(* PLC project Unnamed, Unknown Unnamed 1 *)
(* stored: creationDateTime 2022-09-05T09:02:48, modificationDateTime 2022-09-09T09:39:37 *)

FUNCTION_BLOCK my_functionBlock
  VAR
    MYNODE : HMI_NODE;  (* Using HMI_NODE creates node un HMI tree *)
    SOME_INT : HMI_INT;
  END_VAR
  VAR_INPUT
    SOME_STRING : HMI_STRING;
  END_VAR
  VAR
    SOME_BOOL : HMI_BOOL;
    SOME_REAL : HMI_REAL;
  END_VAR
  VAR_INPUT
    SOME_INPUT : BOOL;
  END_VAR
  VAR_OUTPUT
    SOME_OUTPUT : BOOL;
  END_VAR

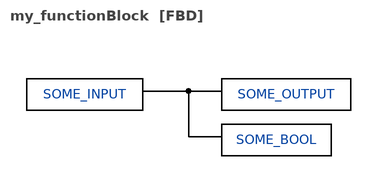
(* FBD diagram, written out as Structured Text *)
SOME_OUTPUT := SOME_INPUT;
SOME_BOOL := SOME_INPUT;
END_FUNCTION_BLOCK

PROGRAM program0
  VAR
    LOGGER0 : LOGGER;
    ENTERING_PAGE : HMI_BOOL;
    LEVEL : LOGLEVEL := DEBUG;
  END_VAR
  VAR_EXTERNAL
    CURRENT_PAGE_0 : HMI_STRING;
  END_VAR
  VAR
    R_TRIG0 : R_TRIG;
    ENABLE_JUMP : HMI_BOOL;
    FB_ZERO : my_functionBlock;
    FB_ONE : my_functionBlock;
    FB_TWO : my_functionBlock;
    FB_THREE : my_functionBlock;
    FB_FOUR : my_functionBlock;
    FB_FIVE : my_functionBlock;
    Enable0 : HMI_BOOL := TRUE;
    Enable1 : HMI_BOOL;
    Enable2 : HMI_BOOL := TRUE;
    Enable3 : HMI_BOOL := TRUE;
    Enable4 : HMI_BOOL;
    Enable5 : HMI_BOOL := TRUE;
  END_VAR
  VAR  (* added by the conversion: wires and edge detectors of the diagram *)
    F_TRIG1 : F_TRIG;
  END_VAR

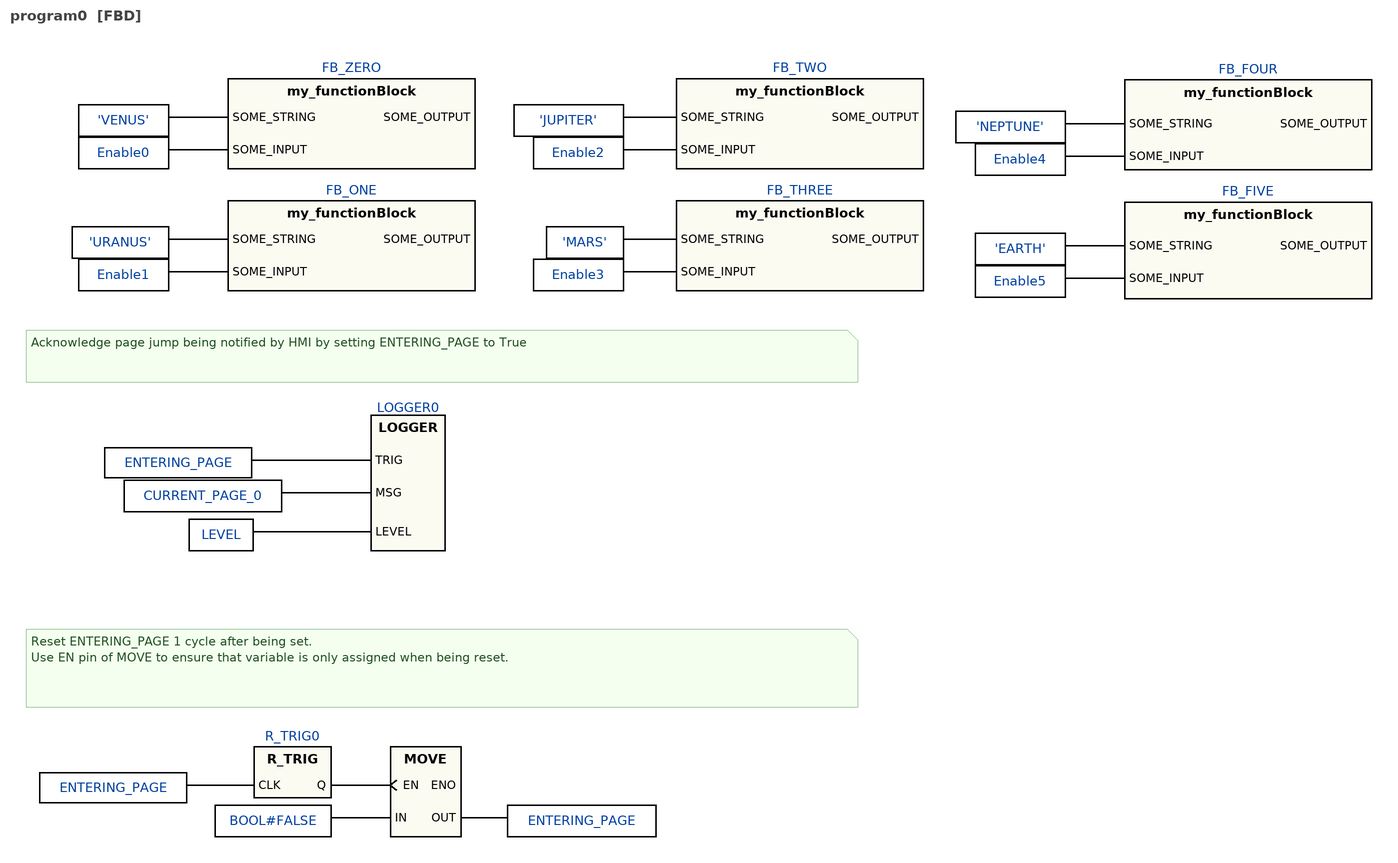
(* FBD diagram, written out as Structured Text *)
(* Acknowledge page jump being notified by HMI by setting ENTERING_PAGE to True *)
(* Reset ENTERING_PAGE 1 cycle after being set. 
Use EN pin of MOVE to ensure that variable is only assigned when being reset. *)
R_TRIG0(CLK := ENTERING_PAGE);
F_TRIG1(CLK := R_TRIG0.Q);
IF F_TRIG1.Q THEN ENTERING_PAGE := BOOL#FALSE; END_IF;
FB_ZERO(SOME_STRING := 'VENUS', SOME_INPUT := Enable0);
FB_TWO(SOME_STRING := 'JUPITER', SOME_INPUT := Enable2);
FB_FOUR(SOME_STRING := 'NEPTUNE', SOME_INPUT := Enable4);
FB_ONE(SOME_STRING := 'URANUS', SOME_INPUT := Enable1);
FB_THREE(SOME_STRING := 'MARS', SOME_INPUT := Enable3);
FB_FIVE(SOME_STRING := 'EARTH', SOME_INPUT := Enable5);
LOGGER0(TRIG := ENTERING_PAGE, MSG := CURRENT_PAGE_0, LEVEL := LEVEL);
END_PROGRAM

CONFIGURATION config
  RESOURCE resource1 ON PLC
    TASK task0(INTERVAL := T#20ms, PRIORITY := 0);
    PROGRAM instance0 WITH task0 : program0;
  END_RESOURCE
END_CONFIGURATION
